FUNCTION_BLOCK CROSSCOMM_PEER_12120F4A7FB80576D (* Service Interface Function Block Type *)
  (* Standard: 61499-2 *)
  (* Version 0.0, 9/22/2017, bababen, nxtControl GmbH, template *)
  PACKAGE Main;
  (* Compiler Cpp nxtControl builtin 1.0 *)
  {SET_ATTRIBUTE(Runtime.FBType.ImplementingType, Runtime.System#DYNGEN_CROSSCOMM_PEER)}
  {SET_ATTRIBUTE(Configuration.GenericFBType.InterfaceParams, Runtime.System#<InterfaceList> <EventOutputs> <Event Name="CNF"> <With Var="LED3" /> <With Var="LED2" /> <With Var="LED1" /> <With Var="LED0" /> </Event> </EventOutputs> <OutputVars> <VarDeclaration Name="LED3" Type="BOOL" /> <VarDeclaration Name="LED2" Type="BOOL" /> <VarDeclaration Name="LED1" Type="BOOL" /> <VarDeclaration Name="LED0" Type="BOOL" /> </OutputVars> </InterfaceList>)}
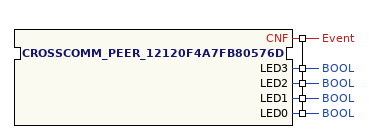
  EVENT_OUTPUT
    CNF WITH LED3, LED2, LED1, LED0;
  END_EVENT
  VAR_OUTPUT
    LED3 : BOOL;
    LED2 : BOOL;
    LED1 : BOOL;
    LED0 : BOOL;
  END_VAR
  EC_STATES
    START;
  END_STATES
END_FUNCTION_BLOCK
